INTERFACE I_SyncUnitTask EXTENDS I_Component

{attribute 'monitoring' := 'call'}
PROPERTY IoDataValid : BOOL
GET
END_GET
END_PROPERTY

{attribute 'monitoring' := 'call'}
PROPERTY IsHotConnect : BOOL
GET
END_GET
END_PROPERTY

{attribute 'monitoring' := 'call'}
PROPERTY PUBLIC SlaveCount : UINT
GET
END_GET
END_PROPERTY

END_INTERFACE

(* stored: Version 1.1.0.1, ProductVersion 3.1.4026.18
   Itf I_SyncUnitTask: Id {c5df68f5-6d75-0adf-17fb-e7b677114901}
   Property IoDataValid: Id {be618f08-b567-4b19-9cb3-bb10f9979a74}
   Get Get: Id {b921a502-e4be-4b28-95fa-3954235f43c9}
   Property IsHotConnect: Id {9c0c794b-7737-0c4b-1807-9ee8ebfdec0c}
   Get Get: Id {74b3a85e-3b20-0806-3417-98d2a1cc8316}
   Property SlaveCount: Id {d965788c-f877-053f-2191-657ba8fcc60f}
   Get Get: Id {6432ecea-f7e2-0f4e-2d8d-45015cbba232} *)
